// TIA Portal V19 export
FUNCTION "TEST SUPPLIES" : Void   // FC19, STL
TITLE = TEST STEAM, AIR AND WATER
{ S7_Optimized_Access := 'TRUE' }
NAME : TESTALL
VERSION : 0.0
// Comment
// stored: AutoNumber false
BEGIN

NETWORK
TITLE = TEST STEAM, AIR AND WATER
      AN    "TANK AUTO";
      R     "DUMMY TEST STEAM";
      R     "DUMMY TEST AIR";
      R     "DUMMY TEST WATER";
      BEC;
      A     "PA0561_Steam";
      JC    M001;
      A     "DUMMY TEST STEAM";
      JC    M002;
      S     "DUMMY TEST STEAM";
      S     "TIM41";
      JU    END;
M002: A     "T 41 DELAY STEAM";
      JC    END;
      S     "ProcessAndPbAlarms"."A"[55];  //A55_NoSteam// no steam
      JU    END;
M001: R     "DUMMY TEST STEAM";
END:  NOP   0;

NETWORK
TITLE = DUMMY TEST AIR SUPPLY
      A     "PA0572_Air";
      JC    c001;
      A     "DUMMY TEST AIR";
      JC    c002;
      S     "DUMMY TEST AIR";
      S     "TIM42";
      JU    c003;
c002: A     "T 42 DELAY AIR";
      JC    c003;
      S     "ProcessAndPbAlarms"."A"[54];  //A54_NoInstrumentAir// no intrument air
      JU    c003;
c001: R     "DUMMY TEST AIR";
c003: NOP   0;
END_FUNCTION
